{attribute 'no_check'}
FUNCTION_BLOCK AX_PARA_SET_ISTPOS (* Datatyp - Set Istpos *)
VAR_INPUT
	Typ														: UDINT := 1; (* 0	NICHT DEFINIERT Wert wird nicht geschrieben
																			1	Absolutposition
																			2	Relativposition
																			5	Moduloposition *)
	Value													: LREAL;
END_VAR
VAR_OUTPUT
END_VAR
VAR
END_VAR

;

END_FUNCTION_BLOCK

(* stored: Version 1.1.0.1, ProductVersion 3.1.4024.12
   POU AX_PARA_SET_ISTPOS: Id {c2d12902-2957-4ada-852c-afb7b4c4641e}, SpecialFunc None *)
